TYPE T_ProductDescription : STRING[48];
END_TYPE

(* stored: Version 1.1.0.1
   DUT T_ProductDescription: Id {e47d7560-c3e0-4edd-ba43-cf19f3629094} *)
